# EPICS substitutions: iocBoot/iocTomoStream_7BM/tomoStream.substitutions
file "$(TOP)/db/tomoStream.template"
{
pattern
{  P,      R, TOMO_SCAN, IMAGE_P, DARK_PVA, FLAT_PVA, RECON_PVA, THETA_PVA}
{7bmb:, TomoStream:, 7bmb:TomoScanStream:, 7bmb:TomoScanStream:PvaPluginPVPrefix, 7bmb:TomoScanStream:StreamDarkFields, 7bmb:TomoScanStream:StreamFlatFields, 7bmb:TomoStream:StreamRecon, 7bmb:TomoScanStream:StreamTheta}
}
